FUNCTION_BLOCK RxDone (* Basic Function Block Type *)
  (* Standard: 61499-2 *)
  (* Version 0.0, 7/16/2026, Schneider Electric, Template *)
  PACKAGE SE.Nereda;
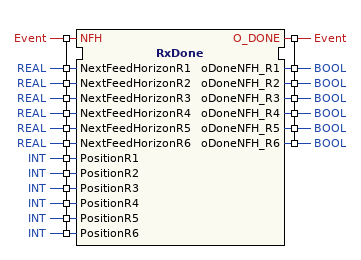
  EVENT_INPUT
    NFH WITH NextFeedHorizonR1, NextFeedHorizonR2, NextFeedHorizonR3, NextFeedHorizonR4, NextFeedHorizonR5, NextFeedHorizonR6, PositionR1, PositionR2, PositionR3, PositionR4, PositionR5, PositionR6;
  END_EVENT
  EVENT_OUTPUT
    O_DONE WITH oDoneNFH_R1, oDoneNFH_R2, oDoneNFH_R3, oDoneNFH_R4, oDoneNFH_R5, oDoneNFH_R6;
  END_EVENT
  VAR_INPUT
    NextFeedHorizonR1 : REAL;
    NextFeedHorizonR2 : REAL;
    NextFeedHorizonR3 : REAL;
    NextFeedHorizonR4 : REAL;
    NextFeedHorizonR5 : REAL;
    NextFeedHorizonR6 : REAL;
    PositionR1 : INT;
    PositionR2 : INT;
    PositionR3 : INT;
    PositionR4 : INT;
    PositionR5 : INT;
    PositionR6 : INT;
  END_VAR
  VAR_OUTPUT
    oDoneNFH_R1 : BOOL;
    oDoneNFH_R2 : BOOL;
    oDoneNFH_R3 : BOOL;
    oDoneNFH_R4 : BOOL;
    oDoneNFH_R5 : BOOL;
    oDoneNFH_R6 : BOOL;
  END_VAR
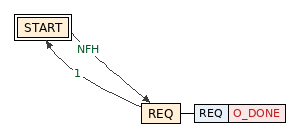
  EC_STATES
    START; (* Initial State *)
    REQ : REQ -> O_DONE; (* Normal execution *)
  END_STATES
  EC_TRANSITIONS
    START TO REQ := NFH;
    REQ TO START := 1;
  END_TRANSITIONS
  ALGORITHM REQ IN ST: (* Normally executed algorithm *)
;
oDoneNFH_R1 := 	PositionR1 > 0 AND NextFeedHorizonR1 <= 0;
oDoneNFH_R2 := 	PositionR2 > 0 AND NextFeedHorizonR2 <= 0;
oDoneNFH_R3 := 	PositionR3 > 0 AND NextFeedHorizonR3 <= 0;
oDoneNFH_R4 := 	PositionR4 > 0 AND NextFeedHorizonR4 <= 0;
oDoneNFH_R5 := 	PositionR5 > 0 AND NextFeedHorizonR5 <= 0;
oDoneNFH_R6 := 	PositionR6 > 0 AND NextFeedHorizonR6 <= 0;
  END_ALGORITHM
END_FUNCTION_BLOCK
